PROGRAM DMC
VAR
	Enable : BOOL;
	el7211 : EL72x1_DMC;
END_VAR

IF Enable THEN
	el7211.Enable();
END_IF









el7211();

END_PROGRAM

(* stored: Version 1.1.0.1, ProductVersion 3.1.4024.9
   POU DMC: Id {27b72ce6-4866-4a8a-9fe4-f9730bfb2d86}, SpecialFunc None *)
